// TIA Portal V20 export
VAR_GLOBAL   // PLC tag table "MC_Constants"
END_VAR
VAR_GLOBAL CONSTANT   // user constants
   DIRA_POSITIVE : Int := 1;   // Orientation direction 1: Positive direction
   DA_DEACTIVATED : Int := 0;   // Dynamic adaption 0: Deactivated
   CS_MCS : Int := 100;   // Coordinate system 100: Machine coordinate system (axis values)
   SM_ACTIVE_DYNAMICS : Int := 0;   // Stop mode 0: Stop with active dynamics
   LC_DEFAULT : DWord := 16#FFFFFFFF;   // LinkConstellation: Default to keep link constellation of kinematics
   CM_CENTER : Int := 1;   // Circle mode 1: "Arc" + "AuxPoint" defines circle center
   ZONE_DEACTIVATION_MODE_SIGNAL : DInt := 3;   // Zone deactivation mode 3: All signal zones
   BM_BLENDING_HIGH : Int := 5;   // Buffer mode 5: Blending with higher velocity
   BM_BUFFERED : Int := 1;   // Buffer mode 1: Standstill between motions
   PC_LONG_RUN_POSITIVE : Int := 2;   // Path choice 2: Longer positive circle segment
   IM_MAX_DYNAMICS : Int := 1;   // Interrupt mode 1: Interrupt with maximum dynamics
   CS_FCS : DInt := 0;   // Coordinate system 0: Flange coordinate system (FCS); Only valid for kinematics zone commands
   CS_TCS : DInt := 1;   // Coordinate system 1: Tool coordinate system (TCS); Only valid for kinematics zone commands
   DA_WITH_VARIABLE_LIMITS : Int := 1;   // Dynamic adaption 1: With segmentation of path
   DIRA_SHORTEST : Int := 3;   // Orientation direction 3: Shortest direction
   CS_OCS3 : Int := 3;   // Coordinate system 3: Object coordinate system 3 (OCS[3])
   CS_OCS1 : Int := 1;   // Coordinate system 1: Object coordinate system 1 (OCS[1])
   CM_RADIUS : Int := 2;   // Circle mode 2: "Radius" + "EndPoint" parameters define the circle segment
   CM_BORDER : Int := 0;   // Circle mode 0: "EndPoint" + "AuxPoint" parameter defines a point on circular path
   SM_MAX_DYNAMICS : Int := 1;   // Stop mode 1: Stop with maximum dynamics
   CP_XZ : Int := 0;   // Circle plane 0: Circle in X-Z plane
   CP_YZ : Int := 1;   // Circle plane 1: Circle in Y-Z plane
   IM_ACTIVE_DYNAMICS : Int := 0;   // Interrupt mode 0: Interrupt with active dynamics
   ZONE_DEACTIVATION_MODE_SPECIFIC : DInt := 0;   // Zone deactivation mode 0: Specific zone index
   BM_BLENDING_LOW : Int := 2;   // Buffer mode 2: Blending with lower velocity
   ZONE_DEACTIVATION_MODE_BLOCKED : DInt := 2;   // Zone deactivation mode 2: All blocked zones
   PC_NEGATIVE : Int := 1;   // Path choice 1: Shorter negative circle segment
   CP_XY : Int := 2;   // Circle plane 2: Circle in X-Y plane
   PM_ABS_ABS : DInt := 1;   // PositionMode 1: Interpretation of cartesian orientation as absolute (only effective for absolute MoveDirect commands)
   DA_WITH_CONSTANT_LIMITS : Int := 2;   // Dynamic adaption 2: No segmentation of path
   CS_OCS2 : Int := 2;   // Coordinate system 2: Object coordinate system 2 (OCS[2])
   CS_JCS : Int := 101;   // Coordinate system 101: Joint coordinate system (joint values)
   ZONE_DEACTIVATION_MODE_WORKSPACE : DInt := 4;   // Zone deactivation mode 4: Currently active workspace zone
   PM_ABS_REL : DInt := 2;   // PositionMode 2: Interpretation of cartesian orientation as relative (only effective for absolute MoveDirect commands)
   DIRA_NEGATIVE : Int := 2;   // Orientation direction 2: Negative direction
   CS_WCS : Int := 0;   // Coordinate system 0: World coordinate system (WCS)
   ZONE_DEACTIVATION_MODE_ALL : DInt := 1;   // Zone deactivation mode 1: All zones
   PC_POSITIVE : Int := 0;   // Path choice 0: Shorter positive circle segment
   PC_LONG_RUN_NEGATIVE : Int := 3;   // Path choice 3: Longer negative circle segment
   DA_DEFAULT : Int := -1;   // Dynamic adaption -1: Use default
END_VAR
